{attribute 'qualified_only'}
{attribute 'strict'}
TYPE E_ProductType:
(
	cube,
	cylinder,
	sphere			
)
;
END_TYPE

(* stored: Version 1.1.0.1, ProductVersion 3.1.4024.13
   DUT E_ProductType: Id {6285f63a-a1f5-4cfa-90c6-fff7032d2f6f} *)
